FUNCTION_BLOCK AOI_Timer
VAR_INPUT
	bEnable: BOOL;
	bReset: BOOL;
END_VAR
VAR_OUTPUT
	diSecond:DINT;
	diMinute: DINT;
	diHour: DINT;
	diTotalSecond: DINT;
	diTotalMinute: DINT;
	diTotalHour: DINT;
END_VAR
VAR
	tonSecond: Ton;
END_VAR

tonSecond(IN:= bEnable AND NOT tonSecond.Q, PT:=T#1000MS , Q=> , ET=> );
IF tonSecond.Q THEN
	diSecond:=diSecond+1;
	diTotalSecond:=diTotalSecond+1;
END_IF

IF diSecond>59 THEN
	diSecond:=0;
	diMinute:=diMinute+1;
	diTotalMinute:=diTotalMinute+1;
END_IF

IF diMinute>59 THEN
	diMinute:=0;
	diHour:=diHour+1;
	diTotalHour:=diTotalHour+1;
END_IF

IF bReset THEN
	diSecond :=0;
	diMinute:=0;
	diHour:=0;
	diTotalSecond:=0;
	diTotalMinute:=0;
	diTotalHour:=0;	
END_IF

END_FUNCTION_BLOCK

(* stored: Version 1.1.0.1, ProductVersion 3.1.4022.16
   POU AOI_Timer: Id {9d53ef77-e013-4fb6-b341-2313db76c901}, SpecialFunc None *)
